# EPICS substitutions: TPGSup/TPG300_switching_functions_rb_AB.substitutions
file TPG300_switching_functions_rb_AB.template {

pattern {PORT, P, Q}

{"\$(PORT)", "\$(P)", "A"}
{"\$(PORT)", "\$(P)", "B"}

}
